(* IEC 61131-3 sources: moqui-plc/agent-skills/output/sessions/isothermal-reactor-001/generated-plc/codesys-applications/IsothermalReactorControl/runtime/component/main/src/main/org/moqui/device, 4 files *)

(* ---- DeviceFacade.dut ---- *)
(*
 * DeviceFacade implementation for managing devices and logical parameters.
 *
 * Naming rules:
 *   deviceName + parameterName or parameterName -> logical signal
 *   deviceName + parameterName or parameterName + Min/Max -> limits
 *
 * All digital signals (boolean) are active-high (positive logic).
 * All durations are expressed in seconds TUnit.
 *)
TYPE DeviceFacade : STRUCT
    (* ========== Analog process/environment parameters ========== *)
    concentrationControllerConcentrationBHighThreshold : REAL; (* Not a physical signal; same documented tooling-gap workaround as tank-level-control-001's threshold parameters (see moqui-device-seed-designer/references/free-standing-parameters.md). Renders as dev.concentrationControllerConcentrationBHighThreshold. Developer-confirmed tuned value 1.2 gmol/liter, set via device-config-survey.yaml, a safety margin below the source material's ~1.266 gmol/liter theoretical maximum (the input-multiplicity zero-process-gain point). *)
    concentrationControllerConcentrationBIn : REAL; (* Physical AI from the C_B composition analyzer. Renders as dev.concentrationControllerConcentrationBIn. Wired manually in InputSignalUpdate (field-engineer-owned). The same manual step also copies this raw value into dev.concentrationControllerFeedback (the ProcessPid instance's feedback input) since that wiring is genuinely site-specific. Instrument span (0-2 gmol/liter) is an assumption giving headroom above the ~1.266 gmol/liter theoretical maximum; confirm against the real analyzer's calibrated range. *)
    concentrationControllerDilutionRateOut : REAL; (* Physical AO representing the dilution rate command (F/V, min^-1), not a 0-100% valve signal (developer-confirmed choice, matches the source material's units and its manipulated-variable excursion constraint directly). Renders as dev.concentrationControllerDilutionRateOut. Converting this to an actual feed valve/pump command using the known constant reactor volume V is manual, in OutputSignalUpdate. *)
    concentrationControllerFeedback : REAL; (* Process feedback. *)
    concentrationControllerOutputActual : REAL; (* Current controller output. *)
    concentrationControllerSetpoint : REAL; (* Process setpoint. *)

    (* ========== Digital process/environment parameters ========== *)
    concentrationControllerActive : BOOL; (* PID active status. *)
    concentrationControllerAtSetpoint : BOOL; (* At setpoint status. *)
    concentrationControllerSleepMode : BOOL; (* Sleep mode active. *)
    concentrationControllerRunCmd : BOOL; (* Drives the Standby<->Run transition (TRUE=Run requested, FALSE=Standby requested), same convention as tank-level-control-001. Renders as dev.concentrationControllerRunCmd. *)

    (* Boolean predicates - computed each scan by MainRuleEngine *)
    concentrationApproachingMax : BOOL; (* Approaching the input-multiplicity zero-process-gain point (threshold confirmed by developer: 1.2 gmol/liter, margin below the source material's ~1.266 gmol/liter theoretical maximum). *)
    concentrationSensorFault : BOOL; (* Analyzer broken-wire/out-of-range detection, 2% margin around an assumed 0-2 gmol/liter instrument span. Generic-fault trigger, same convention as tank-level-control-001's LT sensor check. *)

    (* Operating-mode flags and process timing (mapped from recipe). *)
    (* Project-specific process fields are declared through explicit seed parameters. *)

    (* Main FSM state and transition request/acknowledge commands *)
    status : MainStatus := MainStatus.Standby;
    lastStatus : MainStatus := MainStatus.Standby;
    standbyRequest : BOOL;
    runRequest : BOOL;
    faultRequest : BOOL;
    faultAck : BOOL;

    (* Subsystem FSM states exposed for diagnostics and upstream publication. *)
    (* No subsystem FSMs. *)

    (* ========== Atomic devices ========== *)
    concentrationControllerEnable : BOOL;
    concentrationControllerReset : BOOL;
    concentrationControllerControlSystemId : STRING;
    concentrationControllerControlSystemName : STRING;
    concentrationControllerFeedbackMultiplier : REAL := 1.0;
    concentrationControllerAtSetpointHysteresis : REAL;
    concentrationControllerSetpointMultiplier : REAL := 1.0;
    concentrationControllerSetpointMin : REAL;
    concentrationControllerSetpointMax : REAL;
    concentrationControllerSetpointRampType : RampType := RampType.Linear;
    concentrationControllerSetpointIncreaseTime : TIME := T#0s;
    concentrationControllerSetpointDecreaseTime : TIME := T#0s;
    concentrationControllerSetpointFreezeEnable : BOOL;
    concentrationControllerDeviationInversion : BOOL;
    concentrationControllerOutputMin : REAL;
    concentrationControllerOutputMax : REAL;
    concentrationControllerOutputFreezeEnable : BOOL;
    concentrationControllerGain : REAL := 1.0;
    concentrationControllerIntegrationTime : REAL := 0.0;
    concentrationControllerDerivationTime : REAL := 0.0;
    concentrationControllerOffset : REAL := 0.0;
    concentrationControllerDeadbandRange : REAL;
    concentrationControllerDeadbandDelay : TIME;
    concentrationControllerSleepLevel : REAL := 0.0;
    concentrationControllerSleepDelay : TIME;
    concentrationControllerWakeupDeviation : REAL;
    concentrationControllerWakeupDelay : TIME;
    concentrationControllerSleepBoostLevel : REAL := 0.0;
    concentrationControllerSleepBoostTime : TIME;
    concentrationControllerTrackingMode : BOOL := FALSE;
    concentrationControllerTrackingRef : REAL := 0.0;
    concentrationControllerTickTime : TIME := T#10ms;
    concentrationControllerSetpointEpsilon : REAL := 0.000001;
    concentrationController : ProcessPid;

    (* Signal management - centralised fault / alarm / warning engine *)
    signalMgmt : SignalMgmt;
END_STRUCT END_TYPE

(* ---- IOFacade.dut ---- *)
(*
 * IOFacade implementation for managing physical devices and input/output signals/terminals.
 * Input/Output physical terminals naming rules.
 * From each value of the Parameter entity 3 signals will be generated, according to the following naming convention:
 *     deviceName + parameterName or parameterName + physicalAddress (e.g.: Channel + PhysicalAddress for Modbus)
 *     deviceName + parameterName or parameterName + Min/Max + physicalAddress (e.g.: Channel + PhysicalAddress for Modbus)
 *
 * The physicalAdddress suffix will have the following syntax:
 *    %<memory area prefix> ( <size prefix> )? <memory position>
 * where
 *    <memory area prefix> : I | Q | M
 *    <size prefix> : X | B | W | D
 *    <memory position> : <number> ( .<number> )* (* Depends on the target system *)
 *
 * An alternative is to use semantic signal naming rules.
 *)
TYPE IOFacade : STRUCT
    (* ========== Phyisical Input Terminals/Signals ========== *)
    (* No physical input declarations derived; device-tree binding remains manual. *)

    (* ========== Phyisical Output Terminals/Signals ========== *)
    cbSetpoint : WORD; (* ISOTHERMALREACTORCONTROL_PLC_LiveParametersWrite | moqui/isothermal-reactor/parameters/live *)
END_STRUCT END_TYPE

(* Generation notes:
 * - This file is auto-generable from DeviceRequestItem metadata or from naming conventions.
 * - The logical-to-physical mapping remains outside this template and stays manual in V1.
 *
 * Questions for the skill/user:
 * 1. Should names come from DeviceRequestItem.requestItemName or from naming conventions?
 * 2. Which physical signals are inputs and which are outputs?
 * 3. What IEC type should be used for each signal?
 * 4. Are there address-based names, semantic names, or both?
 *)

(* ---- DeviceDiagnostics.pou ---- *)
{attribute 'no_assign'}
(* Device diagnostics *)
FUNCTION_BLOCK DeviceDiagnostics
VAR_EXTERNAL
    dev : DeviceFacade;
END_VAR
VAR_INPUT
    operationType : OperatingMode := OperatingMode.Run;
END_VAR
VAR_OUTPUT
    error : BOOL;
END_VAR

error := TRUE;

(* Signal management engine *)
(*
 * Prepare a fresh scan (clears the accumulated output action).
 * Then process each device signal in priority order.
 * ImmediateStop -> faultRequest := TRUE -> Main enters Fault state.
 *)
dev.signalMgmt(operationType := SignalMgmtOperatingMode.Prepare);
dev.signalMgmt.operationType := SignalMgmtOperatingMode.Process;

(* Device faults *)
(* ConcentrationController blocking diagnostics *)
dev.signalMgmt(code := 110, category := SignalCategory.Alarm, outputAction := SignalOutputAction.ImmediateStop, activationCondition := dev.concentrationController.invalidConfig, loggerName := dev.signalMgmt.loggerName);

(* Environmental / safety diagnostics *)
(* Safety logic is external; only modeled fault/stop indications are observed here. *)

error := FALSE;

(* Questions for the skill/user:
 * 1. Which device faults are blocking and must trigger ImmediateStop?
 * 2. For each blocking device, which signal should be monitored:
 *    fault, invalidConfig, cmdError, externalFault, etc.?
 * 3. Which environmental/safety predicates should become alarms?
 * 4. Which predicates are warnings only and should not stop the machine?
 *)

(* ---- DeviceManager.pou ---- *)
{attribute 'no_assign'}
(* Hardware Abstraction Layer (HAL) orchestrator.
 *
 * Drives all physical device FBs once per scan.
 * Main component sets the enable/disable request flags; DeviceManager wires them
 * to the individual Actuator / ProcessPid FBs.
 *
 * Call order within the PLC task:
 *   InputSignalUpdate (updates feedback signals from field)
 *   Main (FSM + DeviceRuleEngine -> sets request flags)
 *   DeviceManager (this block - drives device FBs)
 *   OutputSignalUpdate (maps device outputs to physical terminals)
 *
 * Handshake note (Actuator FBs):
 *   enableRequest / disableRequest are VAR_IN_OUT.  The Actuator FB clears
 *   the flag as its acknowledgment.  Main.pou re-asserts the flag each scan
 *   from dev.xxxEnableRequest, so the handshake is level-triggered.
 *
 * ProcessPid note (ahuFan):
 *   ProcessPid uses a plain BOOL 'enable' input - no VAR_IN_OUT handshake.
 *   Setting enable := FALSE ramps the output to 0 and disables the controller.
 *)
FUNCTION_BLOCK DeviceManager
VAR_EXTERNAL
    clks : Clocks;
    dev : DeviceFacade;
END_VAR
VAR_INPUT
    operationType : OperatingMode := OperatingMode.Run;
END_VAR

(* Atomic device orchestration *)
(* ConcentrationController *)
dev.concentrationController(
    enable := dev.concentrationControllerEnable,
    reset := dev.concentrationControllerReset,
    controlSystemId := dev.concentrationControllerControlSystemId,
    controlSystemName := dev.concentrationControllerControlSystemName,
    feedback := dev.concentrationControllerFeedback,
    feedbackMultiplier := dev.concentrationControllerFeedbackMultiplier,
    setpoint := dev.concentrationControllerSetpoint,
    atSetpointHysteresis := dev.concentrationControllerAtSetpointHysteresis,
    setpointMultiplier := dev.concentrationControllerSetpointMultiplier,
    setpointMin := dev.concentrationControllerSetpointMin,
    setpointMax := dev.concentrationControllerSetpointMax,
    setpointRampType := dev.concentrationControllerSetpointRampType,
    setpointIncreaseTime := dev.concentrationControllerSetpointIncreaseTime,
    setpointDecreaseTime := dev.concentrationControllerSetpointDecreaseTime,
    setpointFreezeEnable := dev.concentrationControllerSetpointFreezeEnable,
    deviationInversion := dev.concentrationControllerDeviationInversion,
    outputMin := dev.concentrationControllerOutputMin,
    outputMax := dev.concentrationControllerOutputMax,
    outputFreezeEnable := dev.concentrationControllerOutputFreezeEnable,
    gain := dev.concentrationControllerGain,
    integrationTime := dev.concentrationControllerIntegrationTime,
    derivationTime := dev.concentrationControllerDerivationTime,
    offset := dev.concentrationControllerOffset,
    deadbandRange := dev.concentrationControllerDeadbandRange,
    deadbandDelay := dev.concentrationControllerDeadbandDelay,
    sleepLevel := dev.concentrationControllerSleepLevel,
    sleepDelay := dev.concentrationControllerSleepDelay,
    wakeupDeviation := dev.concentrationControllerWakeupDeviation,
    wakeupDelay := dev.concentrationControllerWakeupDelay,
    sleepBoostLevel := dev.concentrationControllerSleepBoostLevel,
    sleepBoostTime := dev.concentrationControllerSleepBoostTime,
    trackingMode := dev.concentrationControllerTrackingMode,
    trackingRef := dev.concentrationControllerTrackingRef,
    clock := clks.clock10ms,
    tickTime := dev.concentrationControllerTickTime,
    setpointEpsilon := dev.concentrationControllerSetpointEpsilon);

(* Questions for the skill/user:
 * 1. Which atomic devices must be called every scan?
 * 2. For each Actuator, which enableRequest/disableRequest flags drive it?
 * 3. For each ProcessPid, which enable/setpoint/feedback signals drive it?
 * 4. For each Axis or AxisGroup, which command/enable structures are used?
 *)
